PROGRAM POU_WALLLIGHT
VAR
END_VAR

END_PROGRAM

(* stored: Version 1.1.0.1, ProductVersion 3.1.4024.16
   POU POU_WALLLIGHT: Id {840098ec-0897-43ea-8320-196cc3c37fca}, SpecialFunc None *)
